TYPE Intfc_Sender :
STRUCT
	oHandshake				: Handshake_Send;
	iHandshake		 		: Handshake_Receive;
	cReceiverNetId			: STRING;
	cReceiverPort			: UINT;
END_STRUCT
END_TYPE

(* stored: Version 1.1.0.1, ProductVersion 3.1.4022.11
   DUT Intfc_Sender: Id {29483c63-168e-4ce0-a47e-b13634b321b2} *)
